//La FB3 estende la FB1 quindi anche lei implementa l'interfaccia  
//non devo però implementare i metodi get e set delle proprietà
FUNCTION_BLOCK FB3 EXTENDS FB1
VAR_INPUT
	bFlag : bool;
END_VAR
VAR_OUTPUT
END_VAR
VAR
END_VAR

{warning 'add method implementation'}
METHOD returnValue : REAL
//Estensione della funzione base
IF bFlag THEN
	returnValue := SUPER^.returnValue(); //Uso il metodo "padre"
ELSE
	returnValue := 0;		
END_IF
END_METHOD

END_FUNCTION_BLOCK

(* stored: Version 1.1.0.1, ProductVersion 3.1.4022.16
   POU FB3: Id {b0dae3c9-a621-4edc-bc75-2fc7efc12b67}, SpecialFunc None
   Method returnValue: Id {f5547232-e576-4308-b44b-30ac1beffa90} *)
